FUNCTION QUARTERS_TO_LWORD
  (* Standard: 61499-1; Description: Copyright (c) 2024 HR Agrartechnik GmbH This program and the accompanying materials are made available under the terms of the Eclipse Public License 2.0 which is available at https://www.eclipse.org/legal/epl-2.0/ SPDX-License-Identifier: EPL-2.0 *)
  (* Version 1.0, 2024-02-22, franz *)
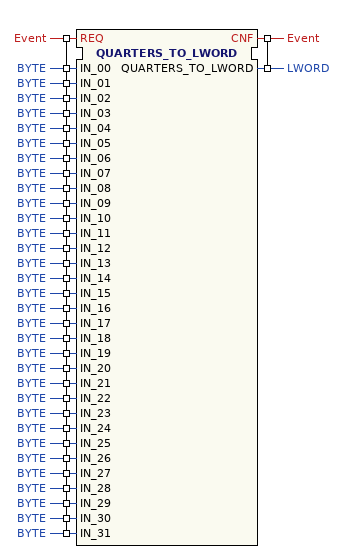
  EVENT_INPUT
    REQ WITH IN_00, IN_01, IN_02, IN_03, IN_04, IN_05, IN_06, IN_07, IN_08, IN_09, IN_10, IN_11, IN_12, IN_13, IN_14, IN_15, IN_16, IN_17, IN_18, IN_19, IN_20, IN_21, IN_22, IN_23, IN_24, IN_25, IN_26, IN_27, IN_28, IN_29, IN_30, IN_31;
  END_EVENT
  EVENT_OUTPUT
    CNF WITH QUARTERS_TO_LWORD;
  END_EVENT
  VAR_INPUT
    IN_00 : BYTE; (* QUARTER BYTE 00 *)
    IN_01 : BYTE; (* QUARTER BYTE 01 *)
    IN_02 : BYTE; (* QUARTER BYTE 02 *)
    IN_03 : BYTE; (* QUARTER BYTE 03 *)
    IN_04 : BYTE; (* QUARTER BYTE 04 *)
    IN_05 : BYTE; (* QUARTER BYTE 05 *)
    IN_06 : BYTE; (* QUARTER BYTE 06 *)
    IN_07 : BYTE; (* QUARTER BYTE 07 *)
    IN_08 : BYTE; (* QUARTER BYTE 08 *)
    IN_09 : BYTE; (* QUARTER BYTE 09 *)
    IN_10 : BYTE; (* QUARTER BYTE 10 *)
    IN_11 : BYTE; (* QUARTER BYTE 11 *)
    IN_12 : BYTE; (* QUARTER BYTE 12 *)
    IN_13 : BYTE; (* QUARTER BYTE 13 *)
    IN_14 : BYTE; (* QUARTER BYTE 14 *)
    IN_15 : BYTE; (* QUARTER BYTE 15 *)
    IN_16 : BYTE; (* QUARTER BYTE 16 *)
    IN_17 : BYTE; (* QUARTER BYTE 17 *)
    IN_18 : BYTE; (* QUARTER BYTE 18 *)
    IN_19 : BYTE; (* QUARTER BYTE 19 *)
    IN_20 : BYTE; (* QUARTER BYTE 20 *)
    IN_21 : BYTE; (* QUARTER BYTE 21 *)
    IN_22 : BYTE; (* QUARTER BYTE 22 *)
    IN_23 : BYTE; (* QUARTER BYTE 23 *)
    IN_24 : BYTE; (* QUARTER BYTE 24 *)
    IN_25 : BYTE; (* QUARTER BYTE 25 *)
    IN_26 : BYTE; (* QUARTER BYTE 26 *)
    IN_27 : BYTE; (* QUARTER BYTE 27 *)
    IN_28 : BYTE; (* QUARTER BYTE 28 *)
    IN_29 : BYTE; (* QUARTER BYTE 29 *)
    IN_30 : BYTE; (* QUARTER BYTE 30 *)
    IN_31 : BYTE; (* QUARTER BYTE 31 *)
  END_VAR
  VAR_OUTPUT
    QUARTERS_TO_LWORD : LWORD;
  END_VAR
  BODY IN ST:
FUNCTION QUARTERS_TO_LWORD : LWORD

VAR_INPUT
	IN_00 : BYTE;    // QUARTER BYTE 00
	IN_01 : BYTE;    // QUARTER BYTE 01
	IN_02 : BYTE;    // QUARTER BYTE 02
	IN_03 : BYTE;    // QUARTER BYTE 03
	IN_04 : BYTE;    // QUARTER BYTE 04
	IN_05 : BYTE;    // QUARTER BYTE 05
	IN_06 : BYTE;    // QUARTER BYTE 06
	IN_07 : BYTE;    // QUARTER BYTE 07
	IN_08 : BYTE;    // QUARTER BYTE 08
	IN_09 : BYTE;    // QUARTER BYTE 09
	IN_10 : BYTE;    // QUARTER BYTE 10
	IN_11 : BYTE;    // QUARTER BYTE 11
	IN_12 : BYTE;    // QUARTER BYTE 12
	IN_13 : BYTE;    // QUARTER BYTE 13
	IN_14 : BYTE;    // QUARTER BYTE 14
	IN_15 : BYTE;    // QUARTER BYTE 15
	IN_16 : BYTE;    // QUARTER BYTE 16
	IN_17 : BYTE;    // QUARTER BYTE 17
	IN_18 : BYTE;    // QUARTER BYTE 18
	IN_19 : BYTE;    // QUARTER BYTE 19
	IN_20 : BYTE;    // QUARTER BYTE 20
	IN_21 : BYTE;    // QUARTER BYTE 21
	IN_22 : BYTE;    // QUARTER BYTE 22
	IN_23 : BYTE;    // QUARTER BYTE 23
	IN_24 : BYTE;    // QUARTER BYTE 24
	IN_25 : BYTE;    // QUARTER BYTE 25
	IN_26 : BYTE;    // QUARTER BYTE 26
	IN_27 : BYTE;    // QUARTER BYTE 27
	IN_28 : BYTE;    // QUARTER BYTE 28
	IN_29 : BYTE;    // QUARTER BYTE 29
	IN_30 : BYTE;    // QUARTER BYTE 30
	IN_31 : BYTE;    // QUARTER BYTE 31
END_VAR

(* this Function combines the 31 QUARTER BYTES to a lword *)
QUARTERS_TO_LWORD := LWORD_QUARTER_ZZ;

QUARTERS_TO_LWORD := QUARTERS_TO_LWORD OR SHL(BYTE_TO_LWORD(IN_31), SHIFT_QUARTER_31);
QUARTERS_TO_LWORD := QUARTERS_TO_LWORD OR SHL(BYTE_TO_LWORD(IN_30), SHIFT_QUARTER_30);
QUARTERS_TO_LWORD := QUARTERS_TO_LWORD OR SHL(BYTE_TO_LWORD(IN_29), SHIFT_QUARTER_29);
QUARTERS_TO_LWORD := QUARTERS_TO_LWORD OR SHL(BYTE_TO_LWORD(IN_28), SHIFT_QUARTER_28);
QUARTERS_TO_LWORD := QUARTERS_TO_LWORD OR SHL(BYTE_TO_LWORD(IN_27), SHIFT_QUARTER_27);
QUARTERS_TO_LWORD := QUARTERS_TO_LWORD OR SHL(BYTE_TO_LWORD(IN_26), SHIFT_QUARTER_26);
QUARTERS_TO_LWORD := QUARTERS_TO_LWORD OR SHL(BYTE_TO_LWORD(IN_25), SHIFT_QUARTER_25);
QUARTERS_TO_LWORD := QUARTERS_TO_LWORD OR SHL(BYTE_TO_LWORD(IN_24), SHIFT_QUARTER_24);
QUARTERS_TO_LWORD := QUARTERS_TO_LWORD OR SHL(BYTE_TO_LWORD(IN_23), SHIFT_QUARTER_23);
QUARTERS_TO_LWORD := QUARTERS_TO_LWORD OR SHL(BYTE_TO_LWORD(IN_22), SHIFT_QUARTER_22);
QUARTERS_TO_LWORD := QUARTERS_TO_LWORD OR SHL(BYTE_TO_LWORD(IN_21), SHIFT_QUARTER_21);
QUARTERS_TO_LWORD := QUARTERS_TO_LWORD OR SHL(BYTE_TO_LWORD(IN_20), SHIFT_QUARTER_20);
QUARTERS_TO_LWORD := QUARTERS_TO_LWORD OR SHL(BYTE_TO_LWORD(IN_19), SHIFT_QUARTER_19);
QUARTERS_TO_LWORD := QUARTERS_TO_LWORD OR SHL(BYTE_TO_LWORD(IN_18), SHIFT_QUARTER_18);
QUARTERS_TO_LWORD := QUARTERS_TO_LWORD OR SHL(BYTE_TO_LWORD(IN_17), SHIFT_QUARTER_17);
QUARTERS_TO_LWORD := QUARTERS_TO_LWORD OR SHL(BYTE_TO_LWORD(IN_16), SHIFT_QUARTER_16);
QUARTERS_TO_LWORD := QUARTERS_TO_LWORD OR SHL(BYTE_TO_LWORD(IN_15), SHIFT_QUARTER_15);
QUARTERS_TO_LWORD := QUARTERS_TO_LWORD OR SHL(BYTE_TO_LWORD(IN_14), SHIFT_QUARTER_14);
QUARTERS_TO_LWORD := QUARTERS_TO_LWORD OR SHL(BYTE_TO_LWORD(IN_13), SHIFT_QUARTER_13);
QUARTERS_TO_LWORD := QUARTERS_TO_LWORD OR SHL(BYTE_TO_LWORD(IN_12), SHIFT_QUARTER_12);
QUARTERS_TO_LWORD := QUARTERS_TO_LWORD OR SHL(BYTE_TO_LWORD(IN_11), SHIFT_QUARTER_11);
QUARTERS_TO_LWORD := QUARTERS_TO_LWORD OR SHL(BYTE_TO_LWORD(IN_10), SHIFT_QUARTER_10);
QUARTERS_TO_LWORD := QUARTERS_TO_LWORD OR SHL(BYTE_TO_LWORD(IN_09), SHIFT_QUARTER_09);
QUARTERS_TO_LWORD := QUARTERS_TO_LWORD OR SHL(BYTE_TO_LWORD(IN_08), SHIFT_QUARTER_08);
QUARTERS_TO_LWORD := QUARTERS_TO_LWORD OR SHL(BYTE_TO_LWORD(IN_07), SHFT_QUARTER_07);
QUARTERS_TO_LWORD := QUARTERS_TO_LWORD OR SHL(BYTE_TO_LWORD(IN_06), SHFT_QUARTER_06);
QUARTERS_TO_LWORD := QUARTERS_TO_LWORD OR SHL(BYTE_TO_LWORD(IN_05), SHFT_QUARTER_05);
QUARTERS_TO_LWORD := QUARTERS_TO_LWORD OR SHL(BYTE_TO_LWORD(IN_04), SHFT_QUARTER_04);
QUARTERS_TO_LWORD := QUARTERS_TO_LWORD OR SHL(BYTE_TO_LWORD(IN_03), SHFT_QUARTER_03);
QUARTERS_TO_LWORD := QUARTERS_TO_LWORD OR SHL(BYTE_TO_LWORD(IN_02), SHFT_QUARTER_02);
QUARTERS_TO_LWORD := QUARTERS_TO_LWORD OR SHL(BYTE_TO_LWORD(IN_01), SHFT_QUARTER_01);
QUARTERS_TO_LWORD := QUARTERS_TO_LWORD OR SHL(BYTE_TO_LWORD(IN_00), SHFT_QUARTER_00);

END_FUNCTION
  END_BODY
END_FUNCTION
